FUNCTION_BLOCK Resource
  (* Version 1.0, 2007-11-27, Goran Cengic, Chalmers *)
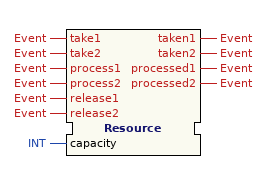
  EVENT_INPUT
    take1;
    take2;
    process1;
    process2;
    release1;
    release2;
  END_EVENT
  EVENT_OUTPUT
    taken1;
    taken2;
    processed1;
    processed2;
  END_EVENT
  VAR_INPUT
    capacity : INT;
  END_VAR
  VAR
    taken : INT;
  END_VAR
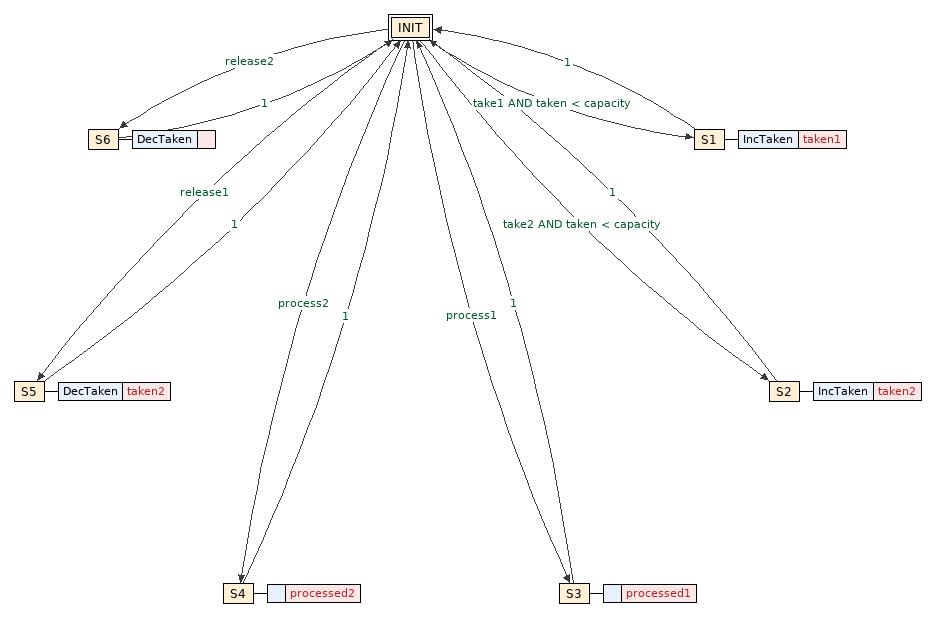
  EC_STATES
    INIT;
    S1 : IncTaken -> taken1;
    S2 : IncTaken -> taken2;
    S3 : -> processed1;
    S4 : -> processed2;
    S5 : DecTaken -> taken2;
    S6 : DecTaken;
  END_STATES
  EC_TRANSITIONS
    INIT TO S1 := take1 AND taken < capacity;
    S1 TO INIT := 1;
    INIT TO S2 := take2 AND taken < capacity;
    S2 TO INIT := 1;
    INIT TO S3 := process1;
    S3 TO INIT := 1;
    INIT TO S4 := process2;
    S4 TO INIT := 1;
    INIT TO S5 := release1;
    S5 TO INIT := 1;
    INIT TO S6 := release2;
    S6 TO INIT := 1;
  END_TRANSITIONS
  ALGORITHM IncTaken IN Java:
taken = (taken + 1) % 3;
  END_ALGORITHM
  ALGORITHM DecTaken IN Java:
taken = (taken + 2) % 3;
  END_ALGORITHM
END_FUNCTION_BLOCK
